// TIA Portal V18 export
ORGANIZATION_BLOCK "Main"   // OB1, LAD, ProgramCycle
TITLE = "Main Program Sweep (Cycle)"
{ S7_Optimized_Access := 'TRUE' }
VERSION : 0.1
// stored: AutoNumber true, IsIECCheckEnabled false, SetENOAutomatically false
BEGIN

REGION Network 1 (SCL)
   "MOTOR_OUTPUT" := ("MOTOR_OUTPUT" OR "MOTOR_START") AND NOT "MOTOR_STOP";
END_REGION
END_ORGANIZATION_BLOCK
